(*
SPDX-FileCopyrightText: © 2026 Oleksandr Tiutyk <trofimich@gmail.com>
SPDX-License-Identifier: MIT
License: https://opensource.org/license/mit
*)

(*!
<summary>Exposes an unsupported-operation exception with a caller-supplied message.</summary>
<description>
Diagnostic string inputs are borrowed only during the call; retained diagnostic text is copied into owned
storage.
</description>
*)
INTERFACE INotSupportedException EXTENDS IGeneralException

(*!
<summary>Raises an unsupported-operation exception with the supplied diagnostic.</summary>
<description>
Long diagnostic strings are borrowed read-only for this call; their references are not retained. Pass
variables or literals, and store computed expressions in local variables before calling. The caller must
supply a nonempty message; this precondition is not checked at runtime.
</description>
*)
METHOD Throw
VAR_INPUT
	sourceNamespaceName : STRING;
	sourceClassName : STRING;
	sourcePOUName : STRING;
	sourcePosition : STRING;
END_VAR
VAR_IN_OUT CONSTANT
	message : ERROR_MESSAGE;
END_VAR
END_METHOD

END_INTERFACE

(* stored: Version 1.1.0.1
   Itf INotSupportedException: Id {b2065534-b81c-4039-bb43-b1dd4c41881c}
   Method Throw: Id {6a642db0-a281-43c5-a141-1a8bc4762080} *)
